(* IEC 61131-3 sources: Industry-PLC-LLM/data/PLCBEAD_repo/PLCBEAD_PLCEmbed-main/PLC-BEAD/Source/GEB/WINDOW2, 1 file *)

(* ---- WINDOW2.ST ---- *)
FUNCTION WINDOW2:BOOL
	VAR_INPUT
		LOW :	REAL;
		IN :	REAL;
		HIGH :	REAL;
	END_VAR
	window2 := (IN <= high) AND (IN >= LOW);
END_FUNCTION

PROGRAM program0
  	VAR
		LOW :	REAL;
		IN :	REAL;
		HIGH :	REAL;
		CEIL5_OUT : BOOL;
	END_VAR

  	CEIL5_OUT := window2(LOW, IN, HIGH);
END_PROGRAM
